// TIA Portal V16 export
// export: Created 2021-06-20T01:36:49.0637285Z, ExportSetting WithDefaults, DisplayName Totally Integrated Automation Portal, DisplayVersion V16 Update 4, DisplayName TIA Portal Version Control Interface, DisplayVersion V16 Update 2, DisplayName TIA Portal Openness, DisplayVersion V16 Update 4, DisplayName STEP 7 Professional, DisplayVersion V16 Update 4, DisplayName STEP 7 Safety, DisplayVersion V16, DisplayName WinCC Advanced, DisplayVersion V16 Update 4
FUNCTION_BLOCK "DoubleAnd"   // FB3, F_FBD
{ S7_Optimized_Access := 'TRUE' }
VERSION : 0.1
// stored: AutoNumber true, IsIECCheckEnabled false, UDAEnableTagReadback false
   VAR_INPUT
      "a" : Bool;
      "b" : Bool;
      c : Bool;
      d : Bool;
   END_VAR
   VAR_OUTPUT
      i : Bool;
      j : Bool;
   END_VAR
BEGIN

REGION Network 1
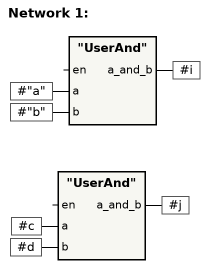
   "UserAnd"("a" := #"a", "b" := #"b", a_and_b => #i);
   "UserAnd"("a" := #c, "b" := #d, a_and_b => #j);
END_REGION
END_FUNCTION_BLOCK
